FUNCTION_BLOCK FBs (* Basic FB with empty ECC *)
  (* Standard: 61499-2 *)
  (* Version 1.0, 2020-10-21, chong *)
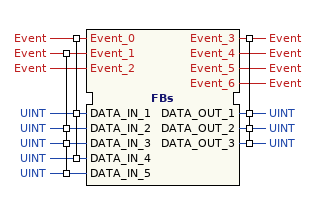
  EVENT_INPUT
    Event_0 WITH DATA_IN_1, DATA_IN_4;
    Event_1 WITH DATA_IN_3, DATA_IN_2, DATA_IN_5;
    Event_2;
  END_EVENT
  EVENT_OUTPUT
    Event_3 WITH DATA_OUT_1, DATA_OUT_2, DATA_OUT_3;
    Event_4;
    Event_5;
    Event_6;
  END_EVENT
  VAR_INPUT
    DATA_IN_1 : UINT;
    DATA_IN_2 : UINT;
    DATA_IN_3 : UINT;
    DATA_IN_4 : UINT;
    DATA_IN_5 : UINT;
  END_VAR
  VAR_OUTPUT
    DATA_OUT_1 : UINT;
    DATA_OUT_2 : UINT;
    DATA_OUT_3 : UINT;
  END_VAR
  EC_STATES
    START; (* Initial State *)
  END_STATES
END_FUNCTION_BLOCK
